(* PLC project PLC, Beckhoff Automation GmbH TwinCAT PLC Control 3.5.13.21 *)
(* stored: creationDateTime 2024-02-17T22:43:08.5303841, modificationDateTime 2024-02-17T22:43:08.5303841 *)

TYPE PBConfig :
STRUCT
	pushDelayTime: TIME;
END_STRUCT
END_TYPE
